// TwinCAT 3 PLC project _16_Proxy
// ProgramVersion: 3.1.4023.0
// libraries:
//   Tc2_Standard, * (Beckhoff Automation GmbH)
//   Tc2_System, * (Beckhoff Automation GmbH)
//   Tc3_Module, * (Beckhoff Automation GmbH)
// project tree:
//   / MAIN.TcPOU, PlcTask.TcTTO
//   Proxy Pattern/ P_Proxy.TcPOU, Proxy.TcPOU, Realsubject.TcPOU (not stored), Subject_Interface.TcIO (not stored)
// (motion and I/O tree: see PLC project 13_decorator)
// real-time tasks:
//   TASK PlcTask: cycle T#10ms, priority 20, ADS port 350
// variable links:

CONFIGURATION _16_Proxy
    RESOURCE PLC ON TwinCAT3
        TASK PlcTask(INTERVAL := T#10ms, PRIORITY := 20);
        PROGRAM MAIN WITH PlcTask : MAIN;
    END_RESOURCE
END_CONFIGURATION

// ---- MAIN.TcPOU
PROGRAM MAIN
VAR
END_VAR

(* 
	GOF 		Provide a surrogate or placeholder for another object to control access to it.
*)
P_Proxy();

END_PROGRAM

// ---- Proxy Pattern/P_Proxy.TcPOU
PROGRAM P_Proxy
VAR
	///Instance of Realsubject but this one is Local to prove on a local and a global object
	localSubjectInstance: Realsubject;
	///Pointer to the local subject. Needed to instantiate its own Proxy. 
	ptrLocalSubject: POINTER TO Realsubject := ADR(localSubjectInstance);
	///Null pointer to the RealSubject class to verify that the other pointers are valid pointers and not null
	ptrNullRealSubject: POINTER TO Realsubject;
	///Pointer needed to create the Connection bridge "Proxy" between the client and the subject 
	ptrProxy: POINTER TO Proxy;
	///Variable to store the password set by the client to perform the connection
	iTempPasswordLocal: INT;
	///Variable to store the INT passed by the client to be SET on the subject
	iSetValueLocal: INT;
	///Boolean value to that gets toggled when the client send a SET request.
	///It is toggled again after the Proxy's response
	bWriteRequest: BOOL;
	///Boolean value to that gets toggled when the client send a GET request.
	///It is toggled again after the Proxy's response
	bReadRequest: BOOL;
	///Variable to store locally if the request was a Write or Read request.
	///TRUE for a Write request and FALSE for a Read request
	bReadWriteLocal: BOOL;
END_VAR
VAR_INPUT
	///Variable to store the response log from the Proxy on a SET request
	sTempSetLog: STRING := 'Waiting for a request';
	///Variable to store the response log from the Proxy on a GET request
	sTempGetLog: STRING := 'Waiting for a request';
	///Variable to store the LAST GET response value locally
	iGetValueLocal: INT;
END_VAR

//The Visualization element can send a GET/SET request with all its parameters.
//Once the request is received by the P_Proxy, the P_Proxy creates the Proxy object to delegate the request and subject's connection to it.
//The default password value for the request is: 1234. It is specified in the static field .iRealPassword of the Proxy class

//If a WRITE or SET request is received
IF	bWriteRequest
	THEN
	//We specify TRUE bReadWriteLocal because it is a SET request
	bReadWriteLocal := TRUE;
	//First we verify if the pointer to RealSubject to be used is a valid pointer
	IF ptrLocalSubject <> ptrNullRealSubject
		//If so, 
		THEN
		//The Proxy object is created with all its parameters passed by the P_Proxy local variables.
		//As there is no "Method Overloading" options is CODESYS (Or at least the constructor cannot be overloaded) the constructor must receive and handle all the possible scenarios
		// .ptrToRealSubject is a Pointer to the RealSubject instance that we try to conncect to
		// .iTempPassword is the password passed by the client in the visualization element
		// .iSetValue is the value passed by the client to be SET on the RealSubject. If the request is a GET request, this value has no effect on the output of the connection.
		// .bReadWrite is the boolean value that specifies if the request is a SET or GET request
		ptrProxy := __NEW( Proxy( ptrToRealSubject := ptrLocalSubject, iTempPassword :=  iTempPasswordLocal, iSetValue := iSetValueLocal, bReadWrite := bReadWriteLocal));
		//Once the Proxy has made the response, the memory is released by deleting the Proxy object
		__DELETE(ptrProxy);
	END_IF
	
	//We delete the local value of last password for security reasons. This way for every request the client must input a password
	iTempPasswordLocal := 0;
	//Once the WRITE request has been handled, we toggle the variable to avoid double requests
	bWriteRequest := FALSE;
END_IF

//If a READ or GET request is received
IF	bReadRequest
	THEN
	//We specify FALSE bReadWriteLocal because it is a GET request
	bReadWriteLocal := FALSE;
	//First we verify if the pointer to RealSubject to be used is a valid pointer
	IF ptrLocalSubject <> ptrNullRealSubject
		//If so,
		THEN
		//The Proxy object is created with all its parameters passed by the P_Proxy local variables.
		//As there is no "Method Overloading" options is CODESYS (Or at least the constructor cannot be overloaded) the constructor must receive and handle all the possible scenarios
		// .ptrToRealSubject is a Pointer to the RealSubject instance that we try to conncect to
		// .iTempPassword is the password passed by the client in the visualization element
		// .iSetValue is the value passed by the client to be SET on the RealSubject. If the request is a GET request, this value has no effect on the output of the connection.
		// .bReadWrite is the boolean value that specifies if the request is a SET or GET request
		ptrProxy := __NEW(Proxy(ptrToRealSubject := ptrLocalSubject, iTempPassword :=  iTempPasswordLocal, iSetValue := 0, bReadWrite := bReadWriteLocal));
		//Once the Proxy has made the response, the memory is released by deleting the Proxy object
		__DELETE(ptrProxy);	
	END_IF
	
	//We delete the local value of last password for security reasons. This way for every request the client must input a password
	iTempPasswordLocal := 0;
	//Once the READ request has been handled, we toggle the variable to avoid double requests
	bReadRequest := FALSE;
END_IF

END_PROGRAM

// ---- Proxy Pattern/Proxy.TcPOU
{attribute 'enable_dynamic_creation' := ''}
FUNCTION_BLOCK Proxy IMPLEMENTS Subject_Interface
VAR
	///Pointer to store the reference to the subject being protected
	refToRealSubject: POINTER TO Realsubject;
	///Last value of password entered by the client in the visualization element
	iTempPassword: INT;
END_VAR
VAR_STAT
	///Default password value for the request to be accepted
	iRealPassword: INT := 1234;
END_VAR

METHOD fb_init
VAR_INPUT
	/// TRUE: the Retain-variables are initialized (reset warm / reset cold)
	bInitRetains: BOOL;
	/// TRUE  the instance will be copied to the copy-code afterward (online change)
	bInCopyCode: BOOL;
	///Pointer to the RealSubject instance 
	ptrToRealSubject: POINTER TO Realsubject;
	///Local variable to store the password passed by the client with the password of the Proxy
	iTempPassword: INT;
	///Local variable to be used in WRITE request, it is the value to be set if the request is accepted
	iSetValue: INT;
	///Boolean value that specifies if the request is a WRITE or READ request
	bReadWrite: BOOL;
END_VAR
//Stores the address of the subject on a field in th Proxy.
THIS^.refToRealSubject := ptrToRealSubject;
//Stores the password value of the client on a field in the Proxy
THIS^.iTempPassword := iTempPassword;

//For security reasons, the Password passed by the client and the Proxi's connection password are compared
IF	THIS^.iTempPassword = THIS^.iRealPassword 
	//If the password sent by the client is correct,
	THEN
	//We verify is the request is a SET or GET request
	IF bReadWrite
		//If the request is a SET request: boolean value TRUE
		THEN
		//The Proxy passes the request to the subject
		THIS^.Set_Method(iSetValue);
		//Once the request is completed, the Proxy responds to the client that the request has been accepted
		P_Proxy.sTempSetLog := 'Request "SET" accepted';
		//If the request is a GET request: boolean value FALSE
		ELSE
		//The Proxy passes the request to the subject
		P_Proxy.iGetValueLocal:= THIS^.Get_Method();
		//Once the request is completed, the Proxy responds to the client that the request has been accepted
		P_Proxy.sTempGetLog := 'Request "GET" accepted';
	END_IF
	
	//If the password sent by the client is incorrect
	ELSE 
	//We verify is the request is a SET or GET request
	IF bReadWrite
		//If the request is a SET request: boolean value TRUE
		THEN
		//The Proxy handles the bad request and response to the client without the subject intervention
		P_Proxy.sTempSetLog := 'Request denied. Wrong password.';
		//If the request is a GET request: boolean value FALSE
		ELSE
		//The Proxy handles the bad request and response to the client without the subject intervention
		P_Proxy.sTempGetLog := 'Request denied. Wrong password.';
	END_IF

END_IF
END_METHOD

METHOD Get_Method : INT
//Calls the Get_Method of the subject through the proxy to read the iProp value of the subject 
// thanks to the pointer reference saved in the field refToRealSubject of the proxy object. 

Get_Method := THIS^.refToRealSubject^.Get_Method();
END_METHOD

METHOD Set_Method
VAR_INPUT
	///Value to be set to the subject passed as an input argument
	num: INT;
END_VAR
//Calls the Set_Method of the subject through the proxy to write the iProp field of the subject 
// thanks to the pointer reference saved in the field refToRealSubject of the proxy object.

THIS^.refToRealSubject^.Set_Method(num);
END_METHOD

END_FUNCTION_BLOCK
